{region '#Template'}
	{attribute 'Version' := '1.2.1.0'}
	{attribute 'Tags' := '"LCID": "1031", "Text": "Universal, Sensor, BI, BV"'}
	{attribute 'Tags' := '"LCID": "1033", "Text": "Universal, Sensor, BI, BV"'}
	{attribute 'Using' := '"Type": "Template", "URI": "EC_AMEV"'}
	{attribute 'Using' := '"Type": "Template", "URI": "BA2_Param"'}
	{attribute 'Description' := '"LCID": "1031", "Text": "Kombination aus BV BI"'}
	{attribute 'Description' := '"LCID": "1033", "Text": "Combination of BV BI"'}
{endregion}	 
FUNCTION_BLOCK FB_BA_CombinationBI_BV EXTENDS FB_BA_View
VAR_INPUT
END_VAR
VAR_INPUT CONSTANT
	Input				: FB_BA_BI_IO;	
	Value				: FB_BA_BV_Op;									
END_VAR
VAR_OUTPUT
	bBI_PrVal			: BOOL;
	bBV_PrVal			: BOOL;	
END_VAR
VAR
END_VAR

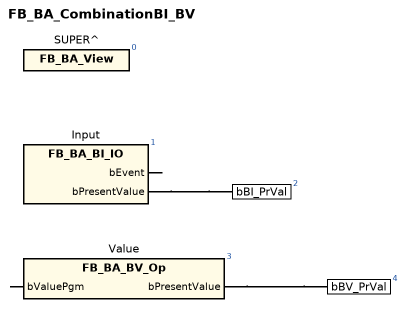
SUPER^(); // FB_BA_View
Input(); // FB_BA_BI_IO
bBI_PrVal := Input.bPresentValue;
Value(); // FB_BA_BV_Op
bBV_PrVal := Value.bPresentValue;

METHOD FB_init : BOOL
VAR_INPUT
	bInitRetains : BOOL; // if TRUE, the retain variables are initialized (warm start / cold start)
	bInCopyCode : BOOL;  // if TRUE, the instance afterwards gets moved into the copy code (online change)
END_VAR
Input.iParent						:= THIS^;
Input.iLabel						:= LblFunctions_Button;	
Input.sObjectName					:= '{Idx=01}';
Input.sDeviceType					:= '';	
Input.bEnOutOfService				:= FALSE;
Input.ePolarity						:= E_BA_Polarity.eReverse;
Input.sActiveText 					:= txtEvent_On;
Input.sInactiveText 				:= txtEvent_Off;
Input.nStateChangeCount				:= 0;
Input.nActiveTimeElapsed			:= 0;
Input.nEventClassID					:= EC_ID.NC80;
Input.stTimeDelay.nToNormal			:= BA2_Param.nDefTimeDelay_ToNormal;
Input.stTimeDelay.nToAbnormal		:= BA2_Param.nDefTimeDelay_ToAbnormal;
Input.bAlarmValue					:= TRUE;
Input.bAcknowledgeRm				:= FALSE;		
Input.aEventTransitionText[1]		:= txtEvent_Off;
Input.aEventTransitionText[2]		:= txtEvent_None;
Input.aEventTransitionText[3]		:= txtEvent_On;
Input.bEventDetectionEnable			:= FALSE;
Input.aEventEnable[1]				:= TRUE;			//	to_offnormal
Input.aEventEnable[2]				:= TRUE;			//	to_fault
Input.aEventEnable[3]				:= TRUE;			//	to_normal
Input.eEnPlantLock					:= E_BA_LockPriority.eNoLock;	

Value.iParent						:= THIS^;		
Value.iLabel 						:= LblFunctions_Button;	
Value.sObjectName					:= '{Idx=02}';	
Value.sActiveText					:= txtEvent_On;
Value.sInactiveText					:= txtEvent_Off;
Value.bValueRm						:= FALSE;
Value.eToggleMode 					:= E_BA_ToggleMode.eSwitch;
END_METHOD

END_FUNCTION_BLOCK

(* stored: Version 1.1.0.1, ProductVersion 3.1.4024.9
   POU FB_BA_CombinationBI_BV: Id {508d4e5b-5bfa-4bc6-bdfb-44d09179e178}, SpecialFunc None
   Method FB_init: Id {c4ebce43-1cde-4c84-af0d-abf189858639} *)
